Fanuc KAREL source: kf00082.KL

PROGRAM KF00082
%STACKSIZE=65535
%PRIORITY=65535
%NOLOCKGROUP
VAR
I : INTEGER
J : INTEGER
X : REAL
Y : REAL
B : BOOLEAN
C : BOOLEAN
TXT : STRING[80]
TXT2 : STRING[80]
AI : ARRAY[4] OF INTEGER
BI : ARRAY[4] OF INTEGER
P : XYZWPR
JP : JOINTPOS9
PF : POSITION
STATUS : INTEGER
-- UNRESOLVED DECLARATIONS (source type spelling not recovered)
-- V1 : TYPE_0x0013 (type_u16=0x0013)
-- V2 : TYPE_0x0013 (type_u16=0x0013)
-- QT : TYPE_0x1100 (type_u16=0x1100)
BEGIN
INIT_QUEUE(QT)
APPEND_QUEUE(3,QT,AI,J,STATUS)
GET_QUEUE(QT,AI,I,STATUS,J)
END KF00082
